(* PLC project Untitled6.project, CODESYS CODESYS V3.5 SP22 Patch 2 *)
(* stored: creationDateTime 2026-07-22T21:18:19.7349617, modificationDateTime 2026-07-22T20:55:16.5590135 *)

PROGRAM PLC_PRG
  VAR
    xStartBtn : BOOL;
    xMotorOnOff : BOOL;
  END_VAR

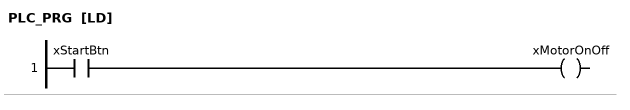
(* LD diagram, written out as Structured Text *)

xMotorOnOff := xStartBtn;
END_PROGRAM
